FUNCTION_BLOCK TRisingEdge
VAR
    R_TRIG1 : R_TRIG;
END_VAR

PROPERTY EdgeDetected : BOOL
GET
EdgeDetected := R_TRIG1.Q;
END_GET
END_PROPERTY

METHOD Test : BOOL
VAR_INPUT
    Value : BOOL;
END_VAR
R_TRIG1(CLK := Value);
Test := R_TRIG1.Q;
END_METHOD

END_FUNCTION_BLOCK

(* stored: Version 1.1.0.1, ProductVersion 3.1.4024.3
   POU TRisingEdge: Id {2c9d8b94-13ec-0fd9-2708-cae11fa383eb}, SpecialFunc None
   Property EdgeDetected: Id {b3438d53-0944-031b-1592-8e49d11dd27f}
   Get Get: Id {e0ce1caa-a188-02ef-083a-3960204bb044}
   Method Test: Id {f11c124b-d542-0c9f-2545-0b5cb4b8356c} *)
